VAR_GLOBAL
	//stTempSensTables	:	ST_TempSensTables;
	VR10	:	ARRAY[1..40,1..2] OF REAL;
	VR11	:	ARRAY[1..40,1..2] OF REAL;
END_VAR

(* stored: Version 1.1.0.1, ProductVersion 3.1.4018.2
   GVL TempConvDat: Id {5679fa5c-7a12-4cb2-aa64-7d14469cc669} *)
